FUNCTION_BLOCK McProcess EXTENDS BaseMcProcess
VAR_INPUT
END_VAR
VAR_OUTPUT
END_VAR
VAR_IN_OUT
END_VAR
VAR
	///At least 1 variable needed because subclass members of an empty class are not exposed by OPC UA (TwinCAT bug!)
	{attribute 'OPC.UA.DA' := '0'}
	testVar: BOOL;
END_VAR

IF do_request THEN
    do_request_result := request();
    do_request := FALSE;
END_IF;
SUPER^();

{attribute 'TcRpcEnable' := '1'}
METHOD request : RequestResults
VAR_INPUT
END_VAR
VAR_OUTPUT
END_VAR
VAR_IN_OUT
END_VAR
VAR
END_VAR
IF THIS^.statuses.enabledStatus.enabled THEN
    THIS^.start();
    request := RequestResults.ACCEPTED;
ELSE
    request := RequestResults.REJECTED;
END_IF;
END_METHOD

{attribute 'TcRpcEnable' := '1'}
METHOD start
VAR_INPUT
END_VAR
VAR_OUTPUT
END_VAR
VAR_IN_OUT
END_VAR
VAR
END_VAR
THIS^.statuses.busyStatus( isBusy := TRUE );
THIS^.statuses.healthStatus( isGood := TRUE );
END_METHOD

END_FUNCTION_BLOCK

(* stored: Version 1.1.0.1, ProductVersion 3.1.4019.2
   POU McProcess: Id {150a0fb9-ce3f-4a89-8cab-e730e66c30a2}, SpecialFunc None
   Method request: Id {34e42db2-1873-43a1-8128-ed35c3075f04}
   Method start: Id {8716ff5d-21d4-48a5-9d6b-a0d2ef5b053b} *)
